(*

.. <legal notes>

legal notes
=================
| SPDX-FileCopyrightText: © 2026 Oleksandr Tiutyk <trofimich@gmail.com>
| SPDX-License-Identifier: LGPL-3.0-only
| For details check: LGPL-3.0-only_

.. _LGPL-3.0-only: https://www.gnu.org/licenses/lgpl-3.0.en.html

.. </legal notes>

*)

TYPE AUTOMATION_ERROR_LOG :
STRUCT
	ShortMessage : Core.ERROR_MESSAGE;
	FullMessage : Core.ERROR_MESSAGE;
	Source : WSTRING(300);
	LocalTimestamp : LDATE_AND_TIME;	
	UtcTimestamp : LDATE_AND_TIME;	
END_STRUCT
END_TYPE

(* stored: Version 1.1.0.1
   DUT AUTOMATION_ERROR_LOG: Id {05878944-5a7a-4222-8e66-d9de192d2acb} *)
